// TwinCAT 3 PLC project PLC
// ProgramVersion: 3.1.4023.0
// libraries:
//   Tc2_Standard, * (Beckhoff Automation GmbH)
//   Tc2_System, * (Beckhoff Automation GmbH)
//   Tc2_Utilities, * (Beckhoff Automation GmbH)
//   Tc3_Module, * (Beckhoff Automation GmbH)
// project tree:
//   DUTs/ stForecast.TcDUT, stWeatherData.TcDUT
//   / PlcTask.TcTTO
//   POUs/ MAIN.TcPOU
// real-time tasks:
//   TASK PlcTask: cycle T#10ms, priority 20, ADS port 350

CONFIGURATION PLC
    RESOURCE PLC ON TwinCAT3
        TASK PlcTask(INTERVAL := T#10ms, PRIORITY := 20);
        PROGRAM MAIN WITH PlcTask : MAIN;
    END_RESOURCE
END_CONFIGURATION

// ---- DUTs/stForecast.TcDUT
TYPE stForecast :
STRUCT
	timeFrom : DT;
	timeTo : DT;
	precipitation_unit : STRING;
	precipitation_value : REAL;
	precipitation_type : STRING;
	windDirection_value : REAL;
	windDirection_name : STRING;
	windSpeed_value : REAL;
	windSpeed_unit : STRING;
	windSpeed_name : STRING;
	temperature_value : REAL;
	temperature_unit : STRING;
	temperature_min : REAL;
	temperature_max : REAL;
	temperature_feel_like : REAL;
	pressure_value : REAL;
	pressure_unit : STRING;
	humidity_value : REAL;
	humidity_UNIT : STRING;
	
END_STRUCT
END_TYPE

// ---- DUTs/stWeatherData.TcDUT
TYPE stWeatherData :
STRUCT
	sunrise : DT;
	sunset : DT;
	Forecast : ARRAY[0..39] OF stForecast;
END_STRUCT
END_TYPE

// ---- POUs/MAIN.TcPOU
PROGRAM MAIN
VAR
	WeatherData : stWeatherData;
	bGetWeatherData : BOOL;
	sysTime : TIMESTRUCT;
	actDateTime : DT;
	fb_LocalSystemTime : FB_LocalSystemTime;
END_VAR

fb_LocalSystemTime(bEnable := TRUE, systemTime => sysTime);
actDateTime := SYSTEMTIME_TO_DT(sysTime);

IF actDateTime > WeatherData.Forecast[0].timeTo THEN
	bGetWeatherData := TRUE;
END_IF

END_PROGRAM
